SUBAPPLICATION Uebung_011a (* Numeric Value Output und BUTTON_PRESS_REPEAT_DONE *)
  (* Standard: 61499-2; Description: Copyright (c) 2023 Meisterschulen am Ostbahnhof This program and the accompanying materials are made available under the terms of the Eclipse Public License 2.0 which is available at https://www.eclipse.org/legal/epl-2.0/ SPDX-License-Identifier: EPL-2.0 *)
  (* Version 1.0, 2023-10-23, Franz Höpfinger, Meisterschulen am Ostbahnhof *)
  IMPORT Uebungen::const::UT::DefaultPool::OutputNumber_N1;
  IMPORT logiBUS::io::DI::logiBUS_DI::Input_I1;
  IMPORT logiBUS::io::DI::logiBUS_DI_Events::BUTTON_PRESS_REPEAT_DONE;
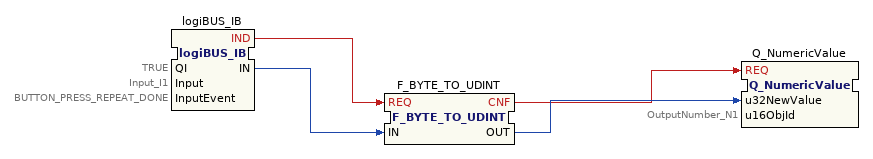
  (* BUTTON_PRESS_REPEAT_DONE: nur am Ende 1 Event BUTTON_PRESS_REPEAT: Während des drückens kommen Events *)
  FBS
    Q_NumericValue : isobus::ut::Q_NumericValue(u16ObjId := OutputNumber_N1);
    logiBUS_IB : logiBUS::io::DI::logiBUS_IB(QI := TRUE, Input := Input_I1, InputEvent := BUTTON_PRESS_REPEAT_DONE);
    F_BYTE_TO_UDINT : iec61131::conversion::F_BYTE_TO_UDINT;
  END_FBS
  EVENT_CONNECTIONS
    logiBUS_IB.IND TO F_BYTE_TO_UDINT.REQ;
    F_BYTE_TO_UDINT.CNF TO Q_NumericValue.REQ;
  END_CONNECTIONS
  DATA_CONNECTIONS
    logiBUS_IB.IN TO F_BYTE_TO_UDINT.IN;
    F_BYTE_TO_UDINT.OUT TO Q_NumericValue.u32NewValue;
  END_CONNECTIONS
END_SUBAPPLICATION
